{attribute 'linkalways'} 
{attribute 'no_explicit_call' := 'This FB is a CLASS and must be accessed using methods or properties'}
{attribute 'enable_dynamic_creation'}
FUNCTION_BLOCK Node_F_VN_CheckIfPointIsInsideContour EXTENDS VisionNode
VAR
    ipContour : _ITcVnContainer;
    aPoint : _TcVnPoint2_REAL;
    fDist : _LREAL(0.0);
    bMeasureDistance : _BOOL(FALSE);
    hrPrev : _HRESULT(S_OK);
	hresult : _HRESULT(S_OK);
END_VAR

METHOD PUBLIC  Clone : I_Node
VAR
	pNode : POINTER TO Node_F_VN_CheckIfPointIsInsideContour;
END_VAR
pNode := __NEW(Node_F_VN_CheckIfPointIsInsideContour);
Clone := pNode^;
END_METHOD

METHOD FB_init : BOOL
VAR_INPUT
	bInitRetains : BOOL; // if TRUE, the retain variables are initialized (warm start / cold start)
	bInCopyCode : BOOL;  // if TRUE, the instance afterwards gets moved into the copy code (online change)
END_VAR
AddInput('ipContour', ipContour);
AddInput('aPoint', aPoint);
AddParameter('bMeasureDistance', bMeasureDistance);
AddInput('hrPrev', hrPrev);
AddOutput('fDist', fDist);
AddOutput('hresult',hresult);
END_METHOD

METHOD PROTECTED OnExecute
hresult.Value := F_VN_CheckIfPointIsInsideContour(
	ipContour := ipContour.Value,
    aPoint := aPoint.Value,
    fDist := fDist.Value,
    bMeasureDistance := bMeasureDistance.Value,
	hrPrev:= hrPrev.Value);
END_METHOD

METHOD PUBLIC PreExecutionCheck
VAR_INPUT
	Check : I_PreExecutionChecks;
END_VAR
Check.IsTrue(ipContour.IsValid, 'ipContour must be a valid container');
Check.IsTrue((ipContour.IsType(TC_GLOBAL_CONST_LIST.ContainerType_Vector_TcVnPoint2_DINT) OR
              ipContour.IsType(TC_GLOBAL_CONST_LIST.ContainerType_Vector_TcVnPoint2_REAL)),
              'ipContour contains incorrect type');
END_METHOD

END_FUNCTION_BLOCK

(* stored: Version 1.1.0.1, ProductVersion 3.1.4026.13
   POU Node_F_VN_CheckIfPointIsInsideContour: Id {9063ca07-e70c-090f-1f69-2ef88f139ef4}, SpecialFunc None
   Folder Constructor: Id {97593cfd-99a5-0e7d-34bd-2892485912ea}
   Method Clone: Id {a0400670-9f4e-0208-1c13-7dc9b77dd06e}
   Method FB_init: Id {b8ef408e-82cc-0f17-20e1-a3005ccc21f3}
   Method OnExecute: Id {5021bd7e-d78c-0032-178b-5e0b0d2d25aa}
   Method PreExecutionCheck: Id {e2c85780-35c5-0d63-1df2-ef94b0ab1916} *)
